// TIA Portal V17 export
// export: Created 2021-12-03T08:13:06.9907696Z, ExportSetting WithDefaults, DisplayName Totally Integrated Automation Portal, DisplayVersion V17, DisplayName TIA Portal Openness, DisplayVersion V17, DisplayName TIA Portal Version Control Interface, DisplayVersion V17, DisplayName STEP 7 Professional, DisplayVersion V17, DisplayName STEP 7 Safety, DisplayVersion V17, DisplayName WinCC Advanced, DisplayVersion V17
FUNCTION_BLOCK "FB_Simulation"   // FB20, FBD
VERSION : 0.1
// stored: AutoNumber false, IsIECCheckEnabled false, UDAEnableTagReadback false
   VAR_TEMP
      T_Circ_BrkCOm : Bool;
      FalseBreaker : Bool;
      FalseConsole : Bool;
      SimConsol : Bool;
      FalseAccelerator : Bool;
      SimAcc : Bool;
      FalseSensor : Bool;
      SimPSConv : Bool;
      FalseSwitch : Bool;
      SimSwitch : Bool;
      SimEnd : Bool;
   END_VAR
BEGIN

REGION Network 1: Симуляция цепей питания сброс
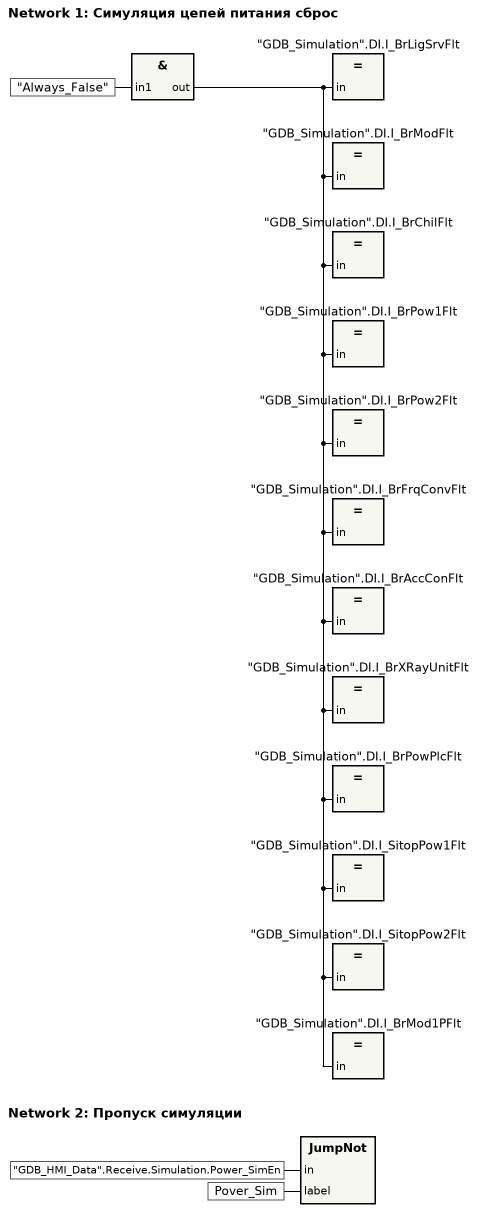
   "GDB_Simulation".DI.I_BrLigSrvFlt := "Always_False";
   "GDB_Simulation".DI.I_BrModFlt := "Always_False";
   "GDB_Simulation".DI.I_BrChilFlt := "Always_False";
   "GDB_Simulation".DI.I_BrPow1Flt := "Always_False";
   "GDB_Simulation".DI.I_BrPow2Flt := "Always_False";
   "GDB_Simulation".DI.I_BrFrqConvFlt := "Always_False";
   "GDB_Simulation".DI.I_BrAccConFlt := "Always_False";
   "GDB_Simulation".DI.I_BrXRayUnitFlt := "Always_False";
   "GDB_Simulation".DI.I_BrPowPlcFlt := "Always_False";
   "GDB_Simulation".DI.I_SitopPow1Flt := "Always_False";
   "GDB_Simulation".DI.I_SitopPow2Flt := "Always_False";
   "GDB_Simulation".DI.I_BrMod1PFlt := "Always_False";
END_REGION

REGION Network 2: Пропуск симуляции
   // no SCL statement known for JumpNot: written as a call
   JumpNot(in := "GDB_HMI_Data".Receive.Simulation.Power_SimEn, label := Pover_Sim);
END_REGION

REGION Network 3: Симуляция цепей питания
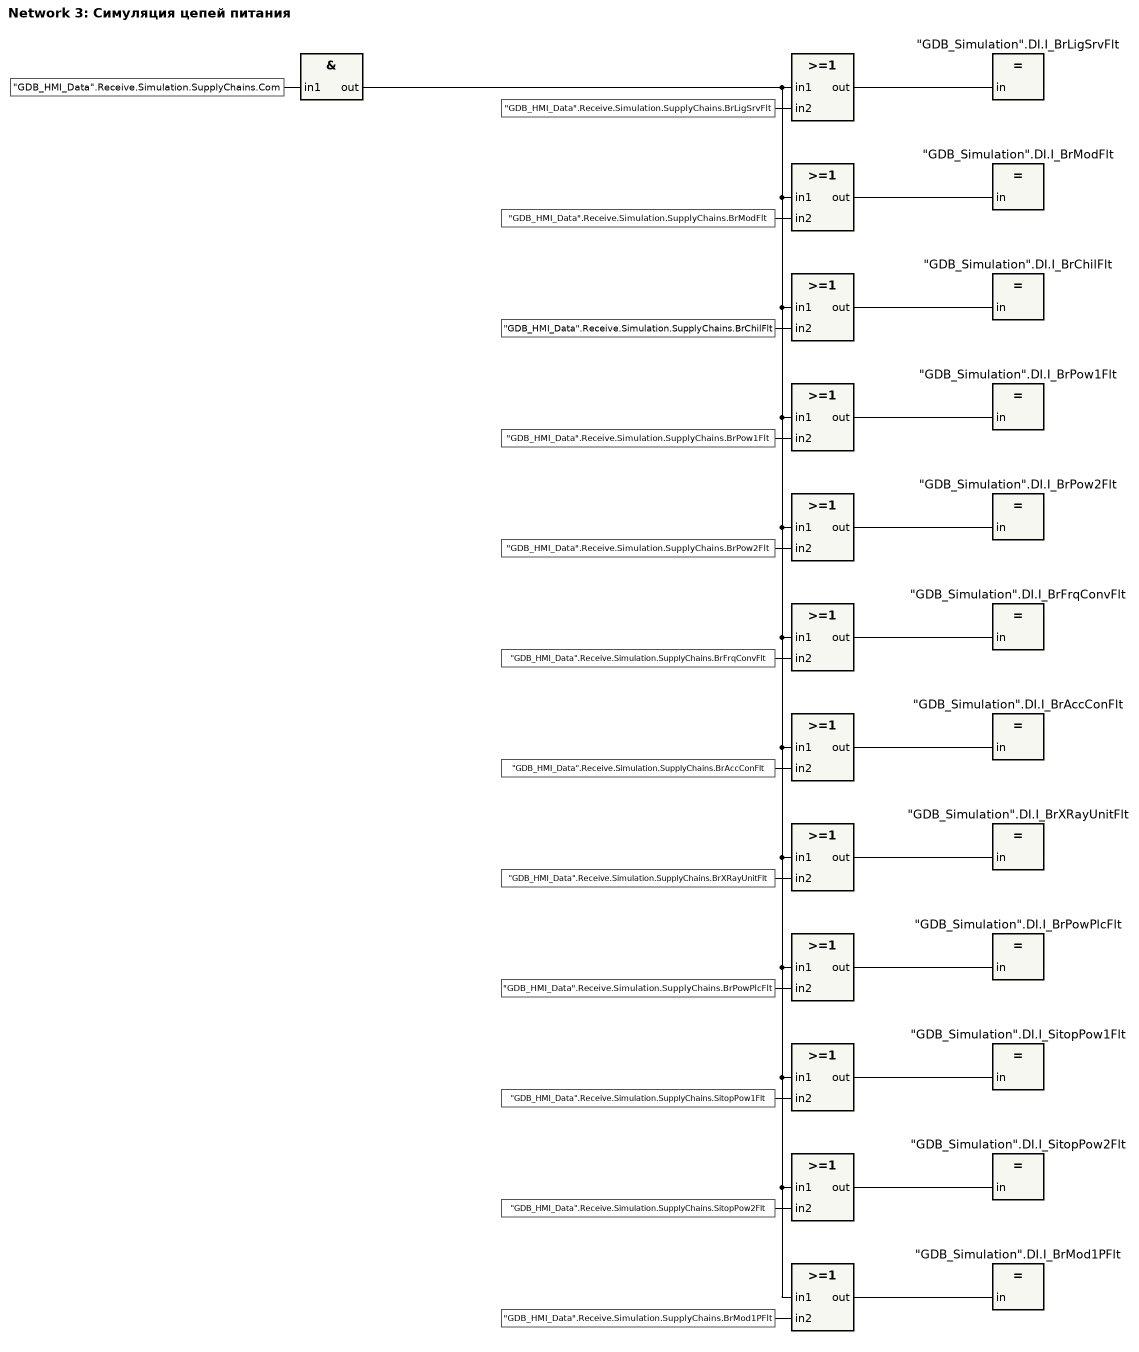
   "GDB_Simulation".DI.I_BrLigSrvFlt := "GDB_HMI_Data".Receive.Simulation.SupplyChains.Com OR "GDB_HMI_Data".Receive.Simulation.SupplyChains.BrLigSrvFlt;
   "GDB_Simulation".DI.I_BrModFlt := "GDB_HMI_Data".Receive.Simulation.SupplyChains.Com OR "GDB_HMI_Data".Receive.Simulation.SupplyChains.BrModFlt;
   "GDB_Simulation".DI.I_BrChilFlt := "GDB_HMI_Data".Receive.Simulation.SupplyChains.Com OR "GDB_HMI_Data".Receive.Simulation.SupplyChains.BrChilFlt;
   "GDB_Simulation".DI.I_BrPow1Flt := "GDB_HMI_Data".Receive.Simulation.SupplyChains.Com OR "GDB_HMI_Data".Receive.Simulation.SupplyChains.BrPow1Flt;
   "GDB_Simulation".DI.I_BrPow2Flt := "GDB_HMI_Data".Receive.Simulation.SupplyChains.Com OR "GDB_HMI_Data".Receive.Simulation.SupplyChains.BrPow2Flt;
   "GDB_Simulation".DI.I_BrFrqConvFlt := "GDB_HMI_Data".Receive.Simulation.SupplyChains.Com OR "GDB_HMI_Data".Receive.Simulation.SupplyChains.BrFrqConvFlt;
   "GDB_Simulation".DI.I_BrAccConFlt := "GDB_HMI_Data".Receive.Simulation.SupplyChains.Com OR "GDB_HMI_Data".Receive.Simulation.SupplyChains.BrAccConFlt;
   "GDB_Simulation".DI.I_BrXRayUnitFlt := "GDB_HMI_Data".Receive.Simulation.SupplyChains.Com OR "GDB_HMI_Data".Receive.Simulation.SupplyChains.BrXRayUnitFlt;
   "GDB_Simulation".DI.I_BrPowPlcFlt := "GDB_HMI_Data".Receive.Simulation.SupplyChains.Com OR "GDB_HMI_Data".Receive.Simulation.SupplyChains.BrPowPlcFlt;
   "GDB_Simulation".DI.I_SitopPow1Flt := "GDB_HMI_Data".Receive.Simulation.SupplyChains.Com OR "GDB_HMI_Data".Receive.Simulation.SupplyChains.SitopPow1Flt;
   "GDB_Simulation".DI.I_SitopPow2Flt := "GDB_HMI_Data".Receive.Simulation.SupplyChains.Com OR "GDB_HMI_Data".Receive.Simulation.SupplyChains.SitopPow2Flt;
   "GDB_Simulation".DI.I_BrMod1PFlt := "GDB_HMI_Data".Receive.Simulation.SupplyChains.Com OR "GDB_HMI_Data".Receive.Simulation.SupplyChains.BrMod1PFlt;
END_REGION

REGION Network 4: Симуляция пультов управления сброс
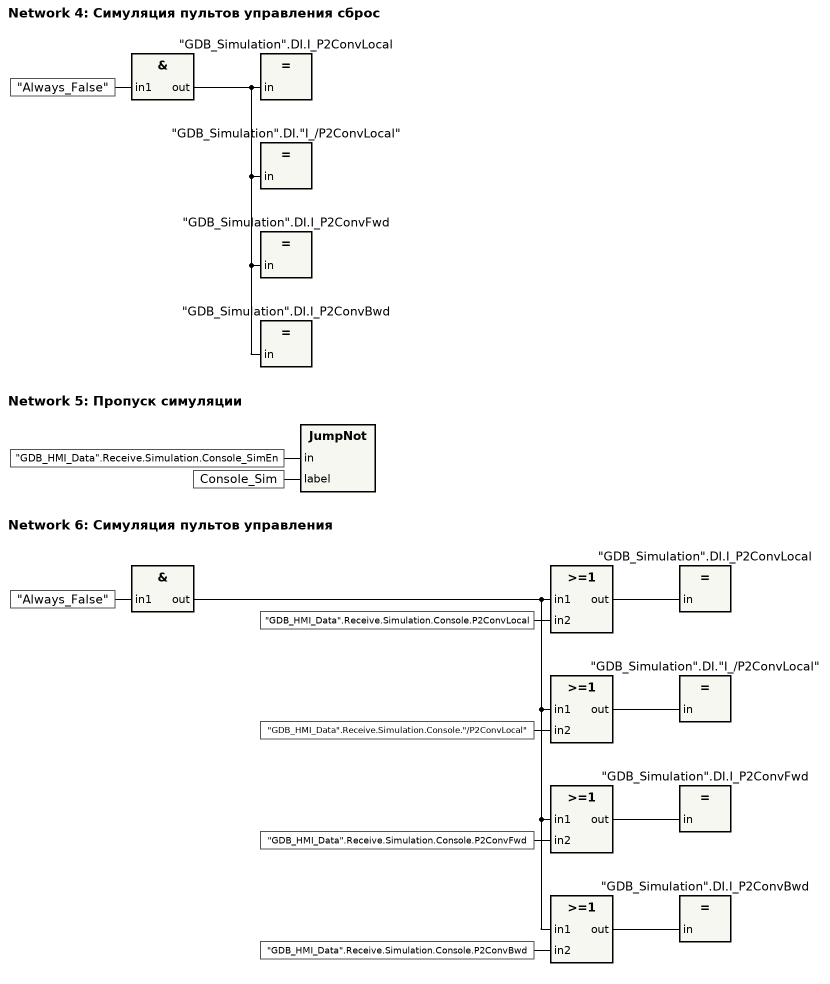
   Pover_Sim:
   "GDB_Simulation".DI.I_P2ConvLocal := "Always_False";
   "GDB_Simulation".DI."I_/P2ConvLocal" := "Always_False";
   "GDB_Simulation".DI.I_P2ConvFwd := "Always_False";
   "GDB_Simulation".DI.I_P2ConvBwd := "Always_False";
END_REGION

REGION Network 5: Пропуск симуляции
   // no SCL statement known for JumpNot: written as a call
   JumpNot(in := "GDB_HMI_Data".Receive.Simulation.Console_SimEn, label := Console_Sim);
END_REGION

REGION Network 6: Симуляция пультов управления
   "GDB_Simulation".DI.I_P2ConvLocal := "Always_False" OR "GDB_HMI_Data".Receive.Simulation.Console.P2ConvLocal;
   "GDB_Simulation".DI."I_/P2ConvLocal" := "Always_False" OR "GDB_HMI_Data".Receive.Simulation.Console."/P2ConvLocal";
   "GDB_Simulation".DI.I_P2ConvFwd := "Always_False" OR "GDB_HMI_Data".Receive.Simulation.Console.P2ConvFwd;
   "GDB_Simulation".DI.I_P2ConvBwd := "Always_False" OR "GDB_HMI_Data".Receive.Simulation.Console.P2ConvBwd;
END_REGION

REGION Network 7: Симуляция сигналов ускорителя сброс
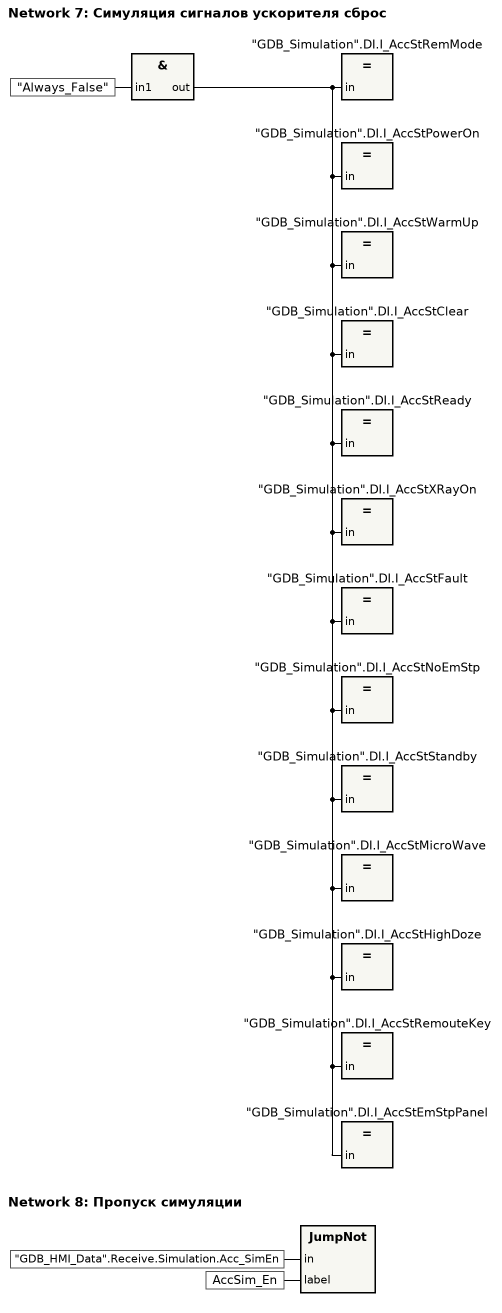
   Console_Sim:
   "GDB_Simulation".DI.I_AccStRemMode := "Always_False";
   "GDB_Simulation".DI.I_AccStPowerOn := "Always_False";
   "GDB_Simulation".DI.I_AccStWarmUp := "Always_False";
   "GDB_Simulation".DI.I_AccStClear := "Always_False";
   "GDB_Simulation".DI.I_AccStReady := "Always_False";
   "GDB_Simulation".DI.I_AccStXRayOn := "Always_False";
   "GDB_Simulation".DI.I_AccStFault := "Always_False";
   "GDB_Simulation".DI.I_AccStNoEmStp := "Always_False";
   "GDB_Simulation".DI.I_AccStStandby := "Always_False";
   "GDB_Simulation".DI.I_AccStMicroWave := "Always_False";
   "GDB_Simulation".DI.I_AccStHighDoze := "Always_False";
   "GDB_Simulation".DI.I_AccStRemouteKey := "Always_False";
   "GDB_Simulation".DI.I_AccStEmStpPanel := "Always_False";
END_REGION

REGION Network 8: Пропуск симуляции
   // no SCL statement known for JumpNot: written as a call
   JumpNot(in := "GDB_HMI_Data".Receive.Simulation.Acc_SimEn, label := AccSim_En);
END_REGION

REGION Network 9: Симуляция сигналов ускорителя
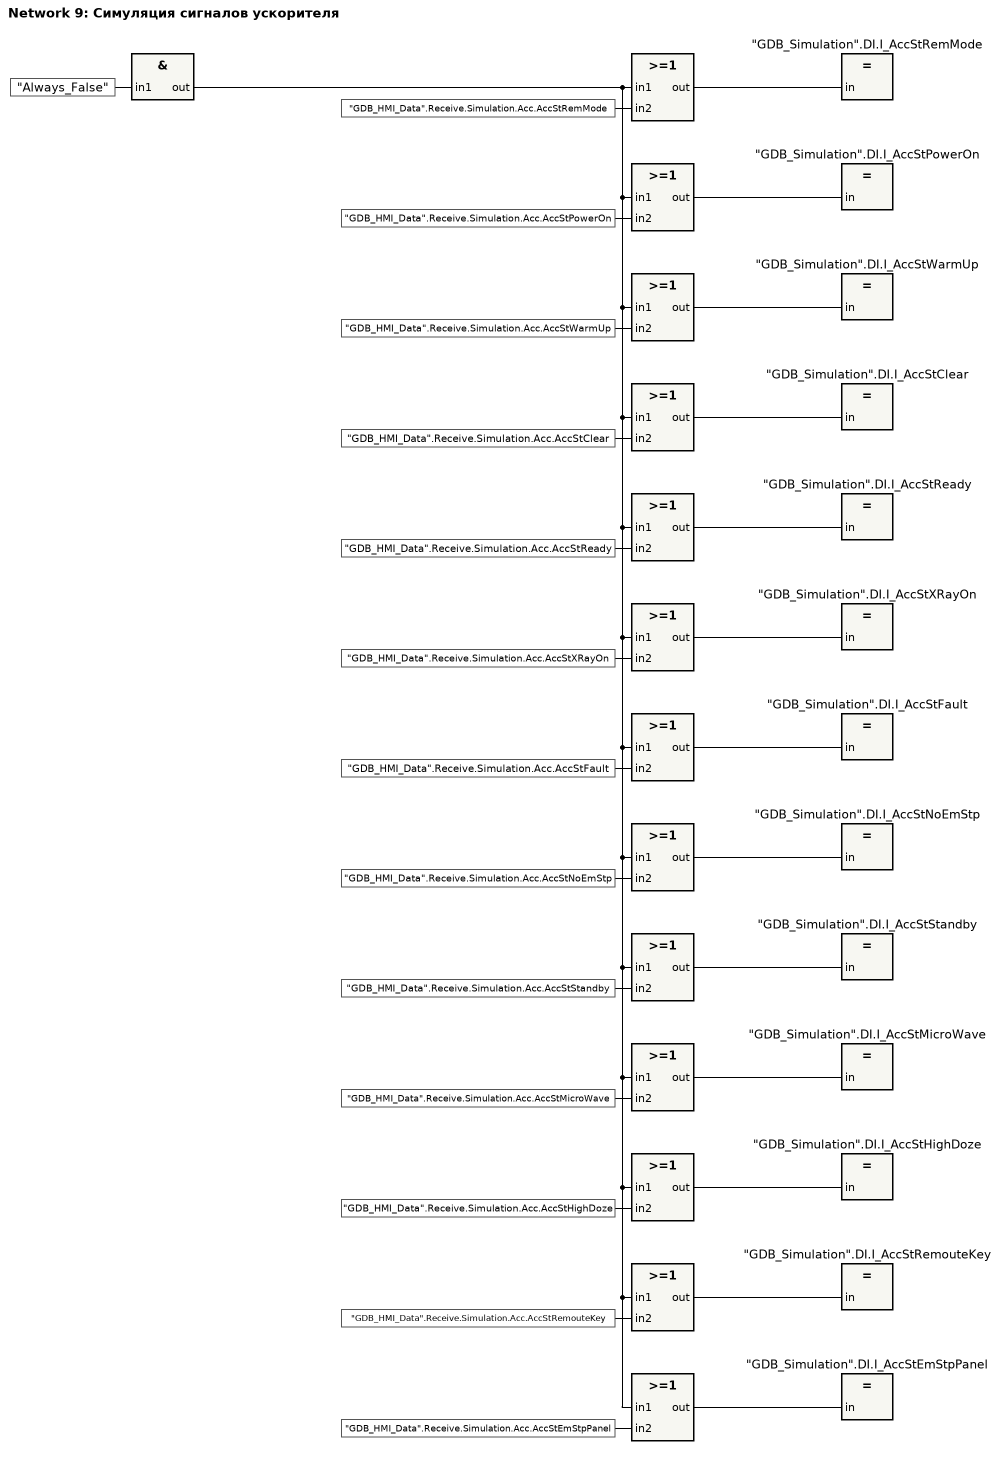
   "GDB_Simulation".DI.I_AccStRemMode := "Always_False" OR "GDB_HMI_Data".Receive.Simulation.Acc.AccStRemMode;
   "GDB_Simulation".DI.I_AccStPowerOn := "Always_False" OR "GDB_HMI_Data".Receive.Simulation.Acc.AccStPowerOn;
   "GDB_Simulation".DI.I_AccStWarmUp := "Always_False" OR "GDB_HMI_Data".Receive.Simulation.Acc.AccStWarmUp;
   "GDB_Simulation".DI.I_AccStClear := "Always_False" OR "GDB_HMI_Data".Receive.Simulation.Acc.AccStClear;
   "GDB_Simulation".DI.I_AccStReady := "Always_False" OR "GDB_HMI_Data".Receive.Simulation.Acc.AccStReady;
   "GDB_Simulation".DI.I_AccStXRayOn := "Always_False" OR "GDB_HMI_Data".Receive.Simulation.Acc.AccStXRayOn;
   "GDB_Simulation".DI.I_AccStFault := "Always_False" OR "GDB_HMI_Data".Receive.Simulation.Acc.AccStFault;
   "GDB_Simulation".DI.I_AccStNoEmStp := "Always_False" OR "GDB_HMI_Data".Receive.Simulation.Acc.AccStNoEmStp;
   "GDB_Simulation".DI.I_AccStStandby := "Always_False" OR "GDB_HMI_Data".Receive.Simulation.Acc.AccStStandby;
   "GDB_Simulation".DI.I_AccStMicroWave := "Always_False" OR "GDB_HMI_Data".Receive.Simulation.Acc.AccStMicroWave;
   "GDB_Simulation".DI.I_AccStHighDoze := "Always_False" OR "GDB_HMI_Data".Receive.Simulation.Acc.AccStHighDoze;
   "GDB_Simulation".DI.I_AccStRemouteKey := "Always_False" OR "GDB_HMI_Data".Receive.Simulation.Acc.AccStRemouteKey;
   "GDB_Simulation".DI.I_AccStEmStpPanel := "Always_False" OR "GDB_HMI_Data".Receive.Simulation.Acc.AccStEmStpPanel;
END_REGION

REGION Network 10: Симуляция фото сенсеров сброс
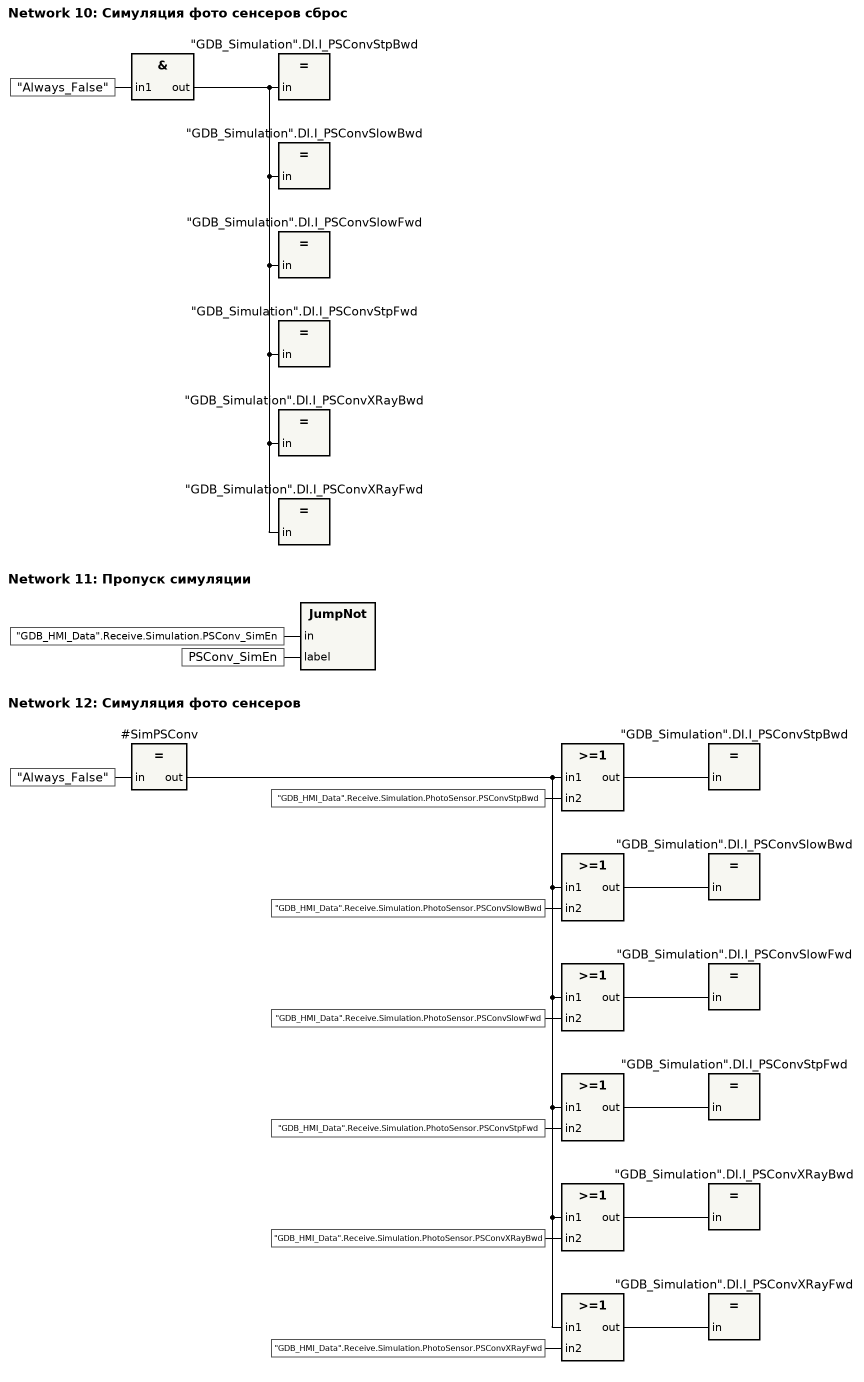
   AccSim_En:
   "GDB_Simulation".DI.I_PSConvStpBwd := "Always_False";
   "GDB_Simulation".DI.I_PSConvSlowBwd := "Always_False";
   "GDB_Simulation".DI.I_PSConvSlowFwd := "Always_False";
   "GDB_Simulation".DI.I_PSConvStpFwd := "Always_False";
   "GDB_Simulation".DI.I_PSConvXRayBwd := "Always_False";
   "GDB_Simulation".DI.I_PSConvXRayFwd := "Always_False";
END_REGION

REGION Network 11: Пропуск симуляции
   // no SCL statement known for JumpNot: written as a call
   JumpNot(in := "GDB_HMI_Data".Receive.Simulation.PSConv_SimEn, label := PSConv_SimEn);
END_REGION

REGION Network 12: Симуляция фото сенсеров
   #SimPSConv := "Always_False";
   "GDB_Simulation".DI.I_PSConvStpBwd := "Always_False" OR "GDB_HMI_Data".Receive.Simulation.PhotoSensor.PSConvStpBwd;
   "GDB_Simulation".DI.I_PSConvSlowBwd := "Always_False" OR "GDB_HMI_Data".Receive.Simulation.PhotoSensor.PSConvSlowBwd;
   "GDB_Simulation".DI.I_PSConvSlowFwd := "Always_False" OR "GDB_HMI_Data".Receive.Simulation.PhotoSensor.PSConvSlowFwd;
   "GDB_Simulation".DI.I_PSConvStpFwd := "Always_False" OR "GDB_HMI_Data".Receive.Simulation.PhotoSensor.PSConvStpFwd;
   "GDB_Simulation".DI.I_PSConvXRayBwd := "Always_False" OR "GDB_HMI_Data".Receive.Simulation.PhotoSensor.PSConvXRayBwd;
   "GDB_Simulation".DI.I_PSConvXRayFwd := "Always_False" OR "GDB_HMI_Data".Receive.Simulation.PhotoSensor.PSConvXRayFwd;
END_REGION

REGION Network 13: Симуляция переключения модулятор чиллер сброс
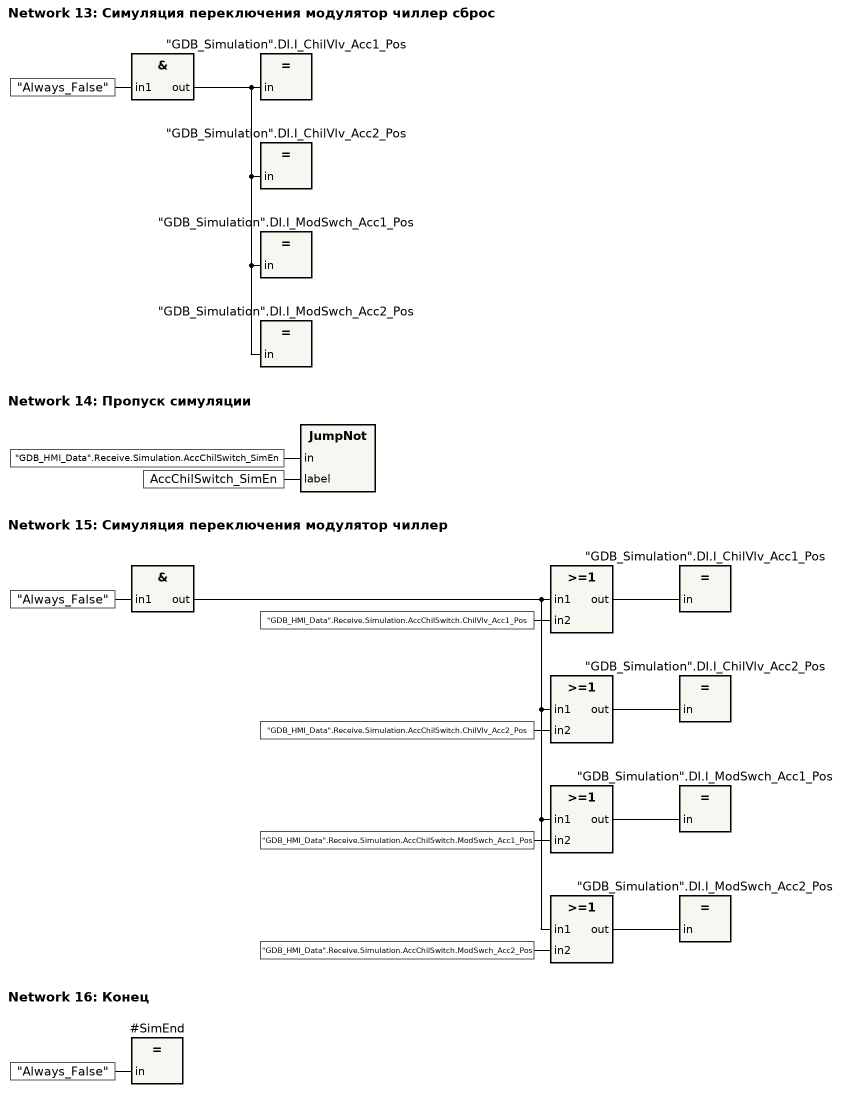
   PSConv_SimEn:
   "GDB_Simulation".DI.I_ChilVlv_Acc1_Pos := "Always_False";
   "GDB_Simulation".DI.I_ChilVlv_Acc2_Pos := "Always_False";
   "GDB_Simulation".DI.I_ModSwch_Acc1_Pos := "Always_False";
   "GDB_Simulation".DI.I_ModSwch_Acc2_Pos := "Always_False";
END_REGION

REGION Network 14: Пропуск симуляции
   // no SCL statement known for JumpNot: written as a call
   JumpNot(in := "GDB_HMI_Data".Receive.Simulation.AccChilSwitch_SimEn, label := AccChilSwitch_SimEn);
END_REGION

REGION Network 15: Симуляция переключения модулятор чиллер
   "GDB_Simulation".DI.I_ChilVlv_Acc1_Pos := "Always_False" OR "GDB_HMI_Data".Receive.Simulation.AccChilSwitch.ChilVlv_Acc1_Pos;
   "GDB_Simulation".DI.I_ChilVlv_Acc2_Pos := "Always_False" OR "GDB_HMI_Data".Receive.Simulation.AccChilSwitch.ChilVlv_Acc2_Pos;
   "GDB_Simulation".DI.I_ModSwch_Acc1_Pos := "Always_False" OR "GDB_HMI_Data".Receive.Simulation.AccChilSwitch.ModSwch_Acc1_Pos;
   "GDB_Simulation".DI.I_ModSwch_Acc2_Pos := "Always_False" OR "GDB_HMI_Data".Receive.Simulation.AccChilSwitch.ModSwch_Acc2_Pos;
END_REGION

REGION Network 16: Конец
   AccChilSwitch_SimEn:
   #SimEnd := "Always_False";
END_REGION
END_FUNCTION_BLOCK
